// Mitsubishi GX Works2 project: 0625(타이머,순차점등)   PLC: Q02/Q02H

PROGRAM MAIN
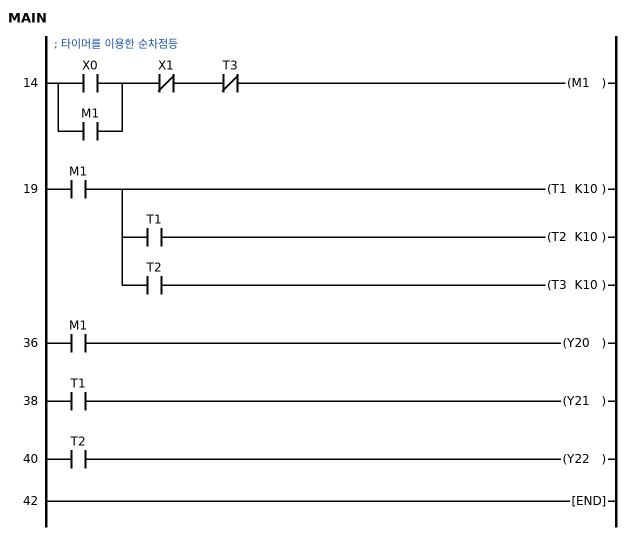
; 타이머를 이용한 순차점등
14    LD      X0
      OR      M1
      ANI     X1
      ANI     T3
      OUT     M1
19    LD      M1
      OUT     T1 K10
      MPS
      AND     T1
      OUT     T2 K10
      MPP
      AND     T2
      OUT     T3 K10
36    LD      M1
      OUT     Y20
38    LD      T1
      OUT     Y21
40    LD      T2
      OUT     Y22
42    END
END_PROGRAM
